(* CODESYS project Horiba.library
   Company: Ziga
   DefaultNamespace: ZigaLibs.Horiba
   Version: 0.0.1.0
   Placeholder: ZigaLibs.Horiba
   Author: Ziga Javornik
   Description: Horiba EtherCAT device imeplementations library.
   Title: ZigaLibs.Horiba

Project tree, tasks and I/O mapping:
  libraries: Tc2_Standard, * (Beckhoff Automation GmbH); Tc2_System, * (Beckhoff Automation GmbH); Tc3_Module, * (Beckhoff Automation GmbH); TcUnit, * (www.tcunit.org); ZigaLibs.Automation, 0.0.1.1 (Ziga); ZigaLibs.Core, 0.0.3.3 (Ziga); ZigaLibs.Logging, 0.0.3.1 (Ziga)
  GVLs/
  SOURCE/
    MFC/
      SEC_ZXX7/
        DUTs/
          data type E_SEC_ZXX7_ActuatorControl
          data type E_SEC_ZXX7_ReadingStep
          data type ST_SEC_ZXX7_ActiveExceptions
          data type ST_SEC_ZXX7_CoeList
          data type ST_SEC_ZXX7_Commands
          data type ST_SEC_ZXX7_Feedback
          data type ST_SEC_ZXX7_Inputs
          data type ST_SEC_ZXX7_Outputs
          data type T_SEC_ZXX7_ActiveExceptionStatus
          data type T_SEC_ZXXX7_RampTime
        POUs/
          function block FB_MFC_SEC_ZXX7 [ST]: FB_init, GasType, GetLogPrefix, RatedFlow, ReadCoe
  TESTS/
    Test suites/
      function block FB_SUT_Tests [ST]: TestXX_Template
    program PRG_TESTS [ST]
*)

// SOURCE/MFC/SEC_ZXX7/DUTs/E_SEC_ZXX7_ActuatorControl
{attribute 'qualified_only'}
{attribute 'strict'}
TYPE E_SEC_ZXX7_ActuatorControl :
(
	FEEDBACK := 0,
	POSITION := 1,
	FULLY_OPEN := 2,
	FULLY_CLOSE := 3,
	FREEZE_POSITION :=4
)USINT;
END_TYPE

// SOURCE/MFC/SEC_ZXX7/DUTs/E_SEC_ZXX7_ReadingStep
{attribute 'qualified_only'}
{attribute 'strict'}
TYPE E_SEC_ZXX7_ReadingStep :
(
	IDLE,
	GAS_TYPE,
	RATED_FLOW
);
END_TYPE

// SOURCE/MFC/SEC_ZXX7/DUTs/ST_SEC_ZXX7_ActiveExceptions
TYPE ST_SEC_ZXX7_ActiveExceptions :
STRUCT
	DeviceWarning		: BOOL;
	DeviceError			: BOOL;
	ManufacturerWarning	: BOOL;
	ManufacturerError	: BOOL;
END_STRUCT
END_TYPE

// SOURCE/MFC/SEC_ZXX7/DUTs/ST_SEC_ZXX7_CoeList
TYPE ST_SEC_ZXX7_CoeList :
STRUCT
	FluidName	: ZigaLibs_Core.ST_CoeEntry_String128 := (Index := 16#900A, Subindex := 16#04);
	Capacity	: ZigaLibs_Core.ST_CoeEntry_REAL := (Index := 16#900A, SubIndex := 16#06);
END_STRUCT
END_TYPE

// SOURCE/MFC/SEC_ZXX7/DUTs/ST_SEC_ZXX7_Commands
TYPE ST_SEC_ZXX7_Commands EXTENDS ST_MfcCommands :
STRUCT
	RampTime	: T_SEC_ZXXX7_RampTime; // Ramp time setpoint in ms	
	Mode		: E_SEC_ZXX7_ActuatorControl;
END_STRUCT
END_TYPE

// SOURCE/MFC/SEC_ZXX7/DUTs/ST_SEC_ZXX7_Feedback
TYPE ST_SEC_ZXX7_Feedback EXTENDS ST_MfcFeedback :
STRUCT
	ActiveExceptions	: ST_SEC_ZXX7_ActiveExceptions;
END_STRUCT
END_TYPE

// SOURCE/MFC/SEC_ZXX7/DUTs/ST_SEC_ZXX7_Inputs
TYPE ST_SEC_ZXX7_Inputs :
STRUCT
	ValvePosition	: REAL;
	ActualFlow		: REAL;
	ExceptionStatus	: T_SEC_ZXX7_ActiveExceptionStatus;
	AmsAddr			: Tc2_System.ST_AmsAddr;
END_STRUCT
END_TYPE

// SOURCE/MFC/SEC_ZXX7/DUTs/ST_SEC_ZXX7_Outputs
TYPE ST_SEC_ZXX7_Outputs :
STRUCT
	FlowSetpoint	: REAL;
	RampTime		: T_SEC_ZXXX7_RampTime;
	ActuatorControl	: E_SEC_ZXX7_ActuatorControl;
END_STRUCT
END_TYPE

// SOURCE/MFC/SEC_ZXX7/DUTs/T_SEC_ZXX7_ActiveExceptionStatus
TYPE T_SEC_ZXX7_ActiveExceptionStatus : USINT; END_TYPE

// SOURCE/MFC/SEC_ZXX7/DUTs/T_SEC_ZXXX7_RampTime
TYPE T_SEC_ZXXX7_RampTime : UDINT; END_TYPE

// SOURCE/MFC/SEC_ZXX7/POUs/FB_MFC_SEC_ZXX7
FUNCTION_BLOCK FB_MFC_SEC_ZXX7 EXTENDS ZigaLibs_Core.FB_HasInstanceNameAndPath
VAR_INPUT
	commands	: ST_SEC_ZXX7_Commands;	// Commands
	updateCoe	: BOOL;	// Reads COE parameters on rising edge
END_VAR

VAR_OUTPUT
	feedback	: ST_SEC_ZXX7_Feedback;	// Feedback
END_VAR

VAR
	_logger			: REFERENCE TO ZigaLibs_Logging.I_Logger;
	_coeList		: ST_SEC_ZXX7_CoeList;
	_exceptionsPrev	: ST_SEC_ZXX7_ActiveExceptions;
	_sb				: ZigaLibs_Core.FB_StringBuilder;
	_init			: BOOL;
	_readRequest	: Tc2_Standard.R_TRIG;
	_ethercatBoxName		: Tc2_System.T_MaxString;
END_VAR

// IO
VAR
	Inputs	AT %I*	: ST_SEC_ZXX7_Inputs;
	Outputs	AT %Q* 	: ST_SEC_ZXX7_Outputs;
END_VAR

IF NOT commands.Enable THEN
	Outputs.ActuatorControl := E_SEC_ZXX7_ActuatorControl.FULLY_CLOSE;
	Outputs.FlowSetpoint := 0;
ELSE
	Outputs.ActuatorControl := commands.Mode;
	Outputs.FlowSetpoint := commands.FlowSetpoint;
	Outputs.RampTime := commands.RampTime;
END_IF

_readRequest(CLK := updateCoe);
IF _readRequest.Q THEN
	_init := FALSE;
END_IF

IF NOT _init THEN
	THIS^.ReadCoe();
END_IF

feedback.ActiveExceptions.DeviceWarning := Inputs.ExceptionStatus.0;
feedback.ActiveExceptions.DeviceError := Inputs.ExceptionStatus.1;
feedback.ActiveExceptions.ManufacturerWarning := Inputs.ExceptionStatus.2;
feedback.ActiveExceptions.ManufacturerError := Inputs.ExceptionStatus.3;
feedback.ValvePosition := Inputs.ValvePosition;
feedback.ActualFlow := inputs.ActualFlow;

// Error logging
IF __ISVALIDREF(_logger) THEN
	IF feedback.ActiveExceptions.DeviceWarning <> _exceptionsPrev.DeviceWarning THEN
		IF feedback.ActiveExceptions.DeviceWarning THEN
			_logger.LogError(_sb.Reset()
				.AddString(THIS^.GetLogPrefix())
				.AddString('Device warning active!')
				.Create());
		ELSE
			_logger.LogInfo(_sb.Reset()
				.AddString(THIS^.GetLogPrefix())
				.AddString('Device warning no longer active!')
				.Create());			
		END_IF
	END_IF
	
	IF feedback.ActiveExceptions.DeviceError <> _exceptionsPrev.DeviceError THEN
		IF feedback.ActiveExceptions.DeviceError THEN
			_logger.LogError(_sb.Reset()
				.AddString(THIS^.GetLogPrefix())
				.AddString('Device error active!')
				.Create());
		ELSE
			_logger.LogInfo(_sb.Reset()
				.AddString(THIS^.GetLogPrefix())
				.AddString('Device error no longer active!')
				.Create());			
		END_IF
	END_IF
	
	IF feedback.ActiveExceptions.ManufacturerWarning <> _exceptionsPrev.ManufacturerWarning THEN
		IF feedback.ActiveExceptions.ManufacturerWarning THEN
			_logger.LogError(_sb.Reset()
				.AddString(THIS^.GetLogPrefix())
				.AddString('Manufacturer warning active!')
				.Create());
		ELSE
			_logger.LogInfo(_sb.Reset()
				.AddString(THIS^.GetLogPrefix())
				.AddString('Manufacturer warning no longer active!')
				.Create());			
		END_IF
	END_IF
	
	IF feedback.ActiveExceptions.ManufacturerError <> _exceptionsPrev.ManufacturerError THEN
		IF feedback.ActiveExceptions.ManufacturerError THEN
			_logger.LogError(_sb.Reset()
				.AddString(THIS^.GetLogPrefix())
				.AddString('Manufacturer error active!')
				.Create());
		ELSE
			_logger.LogInfo(_sb.Reset()
				.AddString(THIS^.GetLogPrefix())
				.AddString('Manufacturer error no longer active!')
				.Create());			
		END_IF
	END_IF
	
END_IF

_exceptionsPrev := feedback.ActiveExceptions;

{attribute 'hide'}
METHOD FB_init : BOOL
VAR_INPUT
	bInitRetains : BOOL; // if TRUE, the retain variables are initialized (warm start / cold start)
	bInCopyCode : BOOL;  // if TRUE, the instance afterwards gets moved into the copy code (online change)
	logger		: REFERENCE TO ZigaLibs_Logging.I_Logger;
END_VAR
_logger REF= logger;
END_METHOD

{attribute 'monitoring' := 'call'}
// Gets the gas type of the MFC
PROPERTY PUBLIC GasType : STRING(128)
GET
GasType := _coeList.FluidName.Value;
END_GET
END_PROPERTY

METHOD PRIVATE GetLogPrefix : T_MaxString
VAR_INPUT
END_VAR
GetLogPrefix := Tc2_Standard.CONCAT(THIS^.InstancePath, ' - ');
END_METHOD

{attribute 'monitoring' := 'call'}
// Gets the rated flow of the MFC
PROPERTY RatedFlow : REAL
GET
RatedFlow := _coeList.Capacity.Value;
END_GET
END_PROPERTY

METHOD PRIVATE ReadCoe
VAR_INPUT
END_VAR
VAR_INST
	fbCoeReadWrite	: ZigaLibs_Core.FB_CoeReadWrite;
	eCoeReadStep	: E_SEC_ZXX7_ReadingStep;
	bError			: BOOL;
END_VAR
CASE eCoeReadStep OF
	E_SEC_ZXX7_ReadingStep.IDLE:
	IF NOT _init THEN
		IF _ethercatBoxName = '' THEN
				_ethercatBoxName := ZigaLibs_Core.EthercatHelper.GetBoxNameByAddress(
					outError := bError,
					PlcRuntimeNetId := '',
					AmsNetId := Inputs.AmsAddr);
			ELSIF _ethercatBoxName <> '' OR bError THEN
				eCoeReadStep := E_SEC_ZXX7_ReadingStep.GAS_TYPE;
				IF __ISVALIDREF(_logger) THEN
					IF NOT bError THEN
						_logger.LogInfo(message := _sb.Reset()	
							.AddString(str := THIS^.GetLogPrefix())
							.AddString(str := 'Reading CoE parameters for Horiba device ')
							.AddWithDblQuotationMarks(str := _ethercatBoxName)
							.AddString(str := '...')
							.Create());
					ELSE
						_logger.LogInfo(message := _sb.Reset()	
							.AddString(str := THIS^.GetLogPrefix())
							.AddString(str := 'Reading CoE parameters for Horiba device ')
							.AddWithDblQuotationMarks(str := '<Error reading EC box name>')
							.AddString(str := '...')
							.Create());
					END_IF
	
				END_IF
			END_IF
		END_IF
		
	E_SEC_ZXX7_ReadingStep.GAS_TYPE:
		IF fbCoeReadWrite.ReadAny(
				CoeEntry := ADR(_CoeList.FluidName),
				Value := _CoeList.FluidName.Value,
				SlaveAddr := Inputs.AmsAddr)
		THEN
			IF __ISVALIDREF(_logger) THEN
				_logger.LogInfo(_sb.Reset()
					.AddString(THIS^.GetLogPrefix())
					.AddString(' - MFC fluid type is ')
					.AddWithDblQuotationMarks(_coeList.FluidName.Value)
					.Create());
			END_IF
			
			eCoeReadStep := E_SEC_ZXX7_ReadingStep.RATED_FLOW;
		END_IF
		
	E_SEC_ZXX7_ReadingStep.RATED_FLOW:
		IF fbCoeReadWrite.ReadAny(
				CoeEntry := ADR(_CoeList.Capacity),
				Value := _CoeList.Capacity.Value,
				SlaveAddr := Inputs.AmsAddr)
		THEN
			IF __ISVALIDREF(_logger) THEN
				_logger.LogInfo(_sb.Reset()
					.AddString(THIS^.GetLogPrefix())
					.AddString(' - MFC rated flow is ')
					.AddAnyReal(_coeList.Capacity.Value, 3, TRUE)
					.AddString(' sccm.')
					.Create());
			END_IF
			
			eCoeReadStep := E_SEC_ZXX7_ReadingStep.IDLE;
			_init := TRUE;
		END_IF
END_CASE
END_METHOD

END_FUNCTION_BLOCK

// TESTS/Test suites/FB_SUT_Tests
// Subject under test
FUNCTION_BLOCK FB_SUT_Tests EXTENDS FB_TestSuite

// Create instance variables that will be accesible for all tests
VAR
END_VAR

// Call your test methods here
TestXX_Template();

METHOD PRIVATE TestXX_Template

(* Instanced variables are VERY useful for writing tests since tests are run in paralel (by default).
By instantiating local variables that are not placed on the same stack as method (values are retained between calls)
you make sure that the SUT is not changed by some other test. *)
VAR_INST
	
END_VAR

// Place temporary variables here
VAR
	
END_VAR
// The name of the test, is the same as method name!
// Use this for paralel unit tests
// TcUnit.TEST('TestXX_Template');

// Use this for running tests in sequence
IF TcUnit.TEST_ORDERED('TestXX_Template') THEN
	// Do your assertions here...
	AssertTrue(
		Condition := FALSE, 
		Message := 'Implement tests!');

	TcUnit.TEST_FINISHED();
END_IF
END_METHOD

END_FUNCTION_BLOCK

// TESTS/PRG_TESTS
PROGRAM PRG_TESTS

(* Instantiate test suites here. Naming convention for tests should be a suffix with _Tests.
Good practice for creating test methods is to end them with _test as well. *)
VAR
	fbSUT_Tests	: FB_SUT_Tests;
END_VAR

// Run tests in parallel
//TcUnit.RUN();

// Run tests in sequence, one after the other.
TcUnit.RUN_IN_SEQUENCE();

END_PROGRAM
